(* PLC project PLC, Beckhoff Automation GmbH TwinCAT PLC Control 3.5.13.21 *)
(* stored: creationDateTime 2024-02-17T22:42:20.9233666, modificationDateTime 2024-02-17T22:42:20.9233666 *)

TYPE LPConfig :
STRUCT
	invert: BOOL;
END_STRUCT
END_TYPE
